(*

## Short summary
This class provides assert statements for 32 bit date and time ``DT``.
It implements the interface `I32BitDtAssertions` 

.. <legal notes>

legal notes
=================
| SPDX-FileCopyrightText: © 2022 ekvip automation GmbH <info@ekvip.de>
| SPDX-License-Identifier: Apache-2.0
| For details check: Apache-2.0_

.. _Apache-2.0: https://www.apache.org/licenses/LICENSE-2.0

.. </legal notes>



*)

{attribute 'reflection'}
FUNCTION_BLOCK INTERNAL DateTimeAssertions32Bit EXTENDS AbstractAssertion IMPLEMENTS I32BitDtAssertions
VAR
END_VAR

(*

## Short summary
This abstract property returns the class name of the concrete object, 
It's for debugging purpose

.. <legal notes>

legal notes
=================
| SPDX-FileCopyrightText: © 2022 ekvip automation GmbH <info@ekvip.de>
| SPDX-License-Identifier: Apache-2.0
| For details check: Apache-2.0_

.. _Apache-2.0: https://www.apache.org/licenses/LICENSE-2.0

.. </legal notes>

*)

PROPERTY className :CNM_AbstractObject.ClassName
GET
className := 'CNM_Assertor.DateTimeAssertions32Bit';
END_GET
END_PROPERTY

(*

## Short summary
This assertion method checks if the current value is equal to the expected value

.. <legal notes>

legal notes
=================
| SPDX-FileCopyrightText: © 2022 ekvip automation GmbH <info@ekvip.de>
| SPDX-License-Identifier: Apache-2.0
| For details check: Apache-2.0_

.. _Apache-2.0: https://www.apache.org/licenses/LICENSE-2.0

.. </legal notes>



*)

METHOD valueIsEqualTo
VAR_INPUT
	(* current value to check *)
	currentValue	:DT;
	(* expected value to compare *)
	expectedValue	:DT;
	(* message if the assertion is false *)
	message			:AssertMessage;
END_VAR
IF (currentValue <> expectedValue) THEN
	THIS^.assertionWasWrong(message, THIS^.getDebugInfo('valueIsEqualTo'));
END_IF
END_METHOD

(*

## Short summary
This assertion method checks if the current value is greater than the less value

.. <legal notes>

legal notes
=================
| SPDX-FileCopyrightText: © 2022 ekvip automation GmbH <info@ekvip.de>
| SPDX-License-Identifier: Apache-2.0
| For details check: Apache-2.0_

.. _Apache-2.0: https://www.apache.org/licenses/LICENSE-2.0

.. </legal notes>



*)

METHOD valueIsGreaterThan
VAR_INPUT
	(* current value to check *)
	currentValue	:DT;
	(* less than lower limit *)
	lessValue		:DT;
	(* message if the assertion is false *)
	message			:AssertMessage;
END_VAR
IF (currentValue <= lessValue) THEN
	THIS^.assertionWasWrong(message, THIS^.getDebugInfo('valueIsGreaterThan'));
END_IF
END_METHOD

(*

## Short summary
This assertion method checks if the current value is inside a limit

**Attention:** 
	limits are included: ``valueIsInRangeOf(dt#1970-01-01-0:0:0, dt#1970-01-01-0:0:0, dt#1970-01-01-0:0:0)``
	is a true assertion

.. <legal notes>

legal notes
=================
| SPDX-FileCopyrightText: © 2022 ekvip automation GmbH <info@ekvip.de>
| SPDX-License-Identifier: Apache-2.0
| For details check: Apache-2.0_

.. _Apache-2.0: https://www.apache.org/licenses/LICENSE-2.0

.. </legal notes>



*)

METHOD valueIsInRangeOf
VAR_INPUT
	(* lower limit for the current value *)
	lowerLimit		:DT;
	(* current value to check *)
	currentValue	:DT;
	(* upper limit for the current value *)
	upperLimit		:DT;
	(* message if the assertion is false *)
	message			:AssertMessage;
END_VAR
IF (
	(currentValue < lowerLimit)
	OR (currentValue > upperLimit)
) THEN
	THIS^.assertionWasWrong(message, THIS^.getDebugInfo('valueIsInRangeOf'));
END_IF
END_METHOD

(*

## Short summary
This assertion method checks if the current value is less than the greater value

.. <legal notes>

legal notes
=================
| SPDX-FileCopyrightText: © 2022 ekvip automation GmbH <info@ekvip.de>
| SPDX-License-Identifier: Apache-2.0
| For details check: Apache-2.0_

.. _Apache-2.0: https://www.apache.org/licenses/LICENSE-2.0

.. </legal notes>



*)

METHOD valueIsLessThan
VAR_INPUT
	(* current value to check *)
	currentValue	:DT;
	(* greater than upper limit *)
	greaterValue	:DT;
	(* message if the assertion is false *)
	message			:AssertMessage;
END_VAR
IF (currentValue >= greaterValue) THEN
	THIS^.assertionWasWrong(message, THIS^.getDebugInfo('valueIsLessThan'));
END_IF
END_METHOD

(*

## Short summary
This assertion method checks if the current value is less than or equal to the maximum value

.. <legal notes>

legal notes
=================
| SPDX-FileCopyrightText: © 2022 ekvip automation GmbH <info@ekvip.de>
| SPDX-License-Identifier: Apache-2.0
| For details check: Apache-2.0_

.. _Apache-2.0: https://www.apache.org/licenses/LICENSE-2.0

.. </legal notes>



*)

METHOD valueIsMax
VAR_INPUT
	(* current value to check *)
	currentValue	:DT;
	(* upper limit for the current value *)
	maximumValue	:DT;
	(* message if the assertion is false *)
	message			:AssertMessage;
END_VAR
IF (currentValue > maximumValue) THEN
	THIS^.assertionWasWrong(message, THIS^.getDebugInfo('valueIsMax'));
END_IF
END_METHOD

(*

## Short summary
This assertion method checks if the current value is greater than or equal to the minimum value

.. <legal notes>

legal notes
=================
| SPDX-FileCopyrightText: © 2022 ekvip automation GmbH <info@ekvip.de>
| SPDX-License-Identifier: Apache-2.0
| For details check: Apache-2.0_

.. _Apache-2.0: https://www.apache.org/licenses/LICENSE-2.0

.. </legal notes>



*)

METHOD valueIsMin
VAR_INPUT
	(* current value to check *)
	currentValue	:DT;
	(* lower limit for the current value *)
	minimumValue	:DT;
	(* message if the assertion is false *)
	message			:AssertMessage;
END_VAR
IF (currentValue < minimumValue) THEN
	THIS^.assertionWasWrong(message, THIS^.getDebugInfo('valueIsMin'));
END_IF
END_METHOD

(*

## Short summary
This assertion method checks if the current value is not equal to the unexpected value

.. <legal notes>

legal notes
=================
| SPDX-FileCopyrightText: © 2022 ekvip automation GmbH <info@ekvip.de>
| SPDX-License-Identifier: Apache-2.0
| For details check: Apache-2.0_

.. _Apache-2.0: https://www.apache.org/licenses/LICENSE-2.0

.. </legal notes>



*)

METHOD valueIsNotEqualTo
VAR_INPUT
	(* current value to check *)
	currentValue	:DT;
	(* unexpected value to compare *)
	unexpectedValue	:DT;
	(* message if the assertion is false *)
	message			:AssertMessage;
END_VAR
IF (currentValue = unexpectedValue) THEN
	THIS^.assertionWasWrong(message, THIS^.getDebugInfo('valueIsNotEqualTo'));
END_IF
END_METHOD

END_FUNCTION_BLOCK

(* stored: Version 1.1.0.1, ProductVersion 3.1.4026.11
   POU DateTimeAssertions32Bit: Id {fb37c652-30ee-4a2a-8584-247bf2cd899c}, SpecialFunc None
   Property className: Id {793b055b-3ba4-4da0-a236-52cb391aaf93}
   Get Get: Id {1ffacb41-a53b-4e2a-bb85-a2f1be4a0c82}
   Method valueIsEqualTo: Id {ca848837-76b8-4d4d-a727-9935ea3cce33}
   Method valueIsGreaterThan: Id {739a04a3-ae5d-436c-a85b-992695e0c425}
   Method valueIsInRangeOf: Id {f561e985-5dce-490e-b772-5a0968033fcf}
   Method valueIsLessThan: Id {35669ee3-6869-49ca-a966-ebc5092c095d}
   Method valueIsMax: Id {281a6825-86a1-4e3c-a3b6-a2064954f9ac}
   Method valueIsMin: Id {d54f0c7a-01a7-41c0-8480-52851fc055c0}
   Method valueIsNotEqualTo: Id {0cc8106c-9082-4d41-98c7-ce8ca3418a0d} *)
